(*
  A start position detection function block dummy.
  A dummy implementation to simulate start triggers at desired positions.
*)
FUNCTION_BLOCK FB_StartPositionDummy EXTENDS FB_BasePrint IMPLEMENTS I_StartPosDetect, I_PrintStatusClient, I_Simulation
VAR_INPUT
  bTrigger                    : BOOL;       // manual trigger
  lPosition                   : DINT;       // current position [SubPx]
  fSpeed                      : LREAL;      // current speed [m/s]
  fResolution                 : LREAL;      // current print resolution [dpi*SubPx]
END_VAR

VAR
  // properties
  _bSim               : BOOL;       // simulatio mode active (PROPERTY)
  _bCreateTrigger     : BOOL;       // create new CT trigger (PROPERTY)
  _nStartPosX0        : DINT;       // create position for CT (absolut) [SubPx] (PROPERTY)
  _bAutoTrigger       : BOOL;       // automatic sheet triggers
  
  // config
  iJobDefinition      : CalmarCompPrint.I_JobDefinition;
  
  // local helper
  rfNewCT             : RF_TRIG;    // trigger new ct
  nSheetLength        : DINT;       // sheet length in [SubPx]
  nSheetGap           : DINT;       // sheet gap in [SubPx]
  nSheetEndPosition   : DINT;       // sheet end position [SubPx]
  nNextSheetPosition  : DINT;       // next trigger location
  fSheetPerHour       : LREAL;      // sheets per hour
  fSheetSpeed         : LREAL;      // [m/min] speed meter per minute
  tCheckTrigger       : TON;
  
  tCurrentTimeStamp   : T_DCTIME64; // get current timestamp
  fCurrentTimeStamp   : LREAL;      // current timestamp
  fSensorTimeStamp    : LREAL;      // sensor timestamp
  fDeltaDistance      : LREAL;      // distance that the substrate moved between the detection and the treatment of the information [m]
END_VAR

VAR PERSISTENT
  // simulation configuration
  fSheetLength   : LREAL := 0.5;    // [m] sheet length (local or per job given)
  fSheetGap      : LREAL := 0.12;   // [m] gap between two sheets
END_VAR

// checks and fixes
IF iJobDefinition = 0 THEN RETURN; END_IF
IF NOT _bSim THEN RETURN; END_IF
IF fSpeed = 0 THEN RETURN; END_IF
IF fSheetLength = 0 THEN fSheetLength := 1; END_IF
IF fResolution = 0 THEN fResolution := 600*32; END_IF

// calculations
fSheetSpeed := fSpeed * 60;  // [m/s] -> [m/min]
nSheetGap := F_MeterToSubPixel(fPosMeter := fSheetGap, fResoSubPx := fResolution);  // [m] -> [SubPx]
fSheetPerHour := (60*60)/((fSheetLength+fSheetGap)/fSpeed);
nSheetLength := F_MeterToSubPixel(fPosMeter := fSheetLength, fResoSubPx := fResolution);  // [mm] -> [SubPx]
nNextSheetPosition := _nStartPosX0 + nSheetLength + nSheetGap; 
tCheckTrigger(PT:=TO_TIME(((fSheetLength+fSheetGap)/fSpeed)*1000));

// internal trigger creation
IF (lPosition - nNextSheetPosition) > 0 AND _bAutoTrigger THEN
  bTrigger := TRUE;
  tCheckTrigger(IN:=FALSE);
  tCheckTrigger(IN:=TRUE);
END_IF

// on trigger
rfNewCT(CLK := bTrigger, RT => _bCreateTrigger);
IF _bCreateTrigger THEN   // new ct created
  bTrigger := FALSE;  // reset trigger
  
  (* Calculate the current and sensor time stamp (keep old code not really necessary because we use current timestamp)*)
  tCurrentTimeStamp := F_GetCurDcTaskTime64();
  fCurrentTimeStamp := (ULINT_TO_LREAL(tCurrentTimeStamp )) / 1_000_000.0; (*in ms*)
  fSensorTimeStamp  := fCurrentTimeStamp;
  fDeltaDistance := (fCurrentTimeStamp - fSensorTimeStamp) * 0.001 * fSpeed;  (*Distance that the substrate moved between the detection and the treatment of the information [m]*)
  
  // sheet start and sheet end pos in [SubPx]
  _nStartPosX0     := lPosition - F_MeterToSubPixel(fPosMeter := fDeltaDistance, fResoSubPx := fResolution);
  nSheetEndPosition := _nStartPosX0 + nSheetLength;
END_IF

PROPERTY bSimEnable : BOOL
GET
bSimEnable := _bSim;
END_GET
SET
_bSim := bSimEnable;
END_SET
END_PROPERTY

(*
  A new container detected.
  NOTE: a pulse only
*)
PROPERTY bStartTrig : BOOL
GET
bStartTrig := _bCreateTrigger;
END_GET
END_PROPERTY

(*
  A valid container detected.
*)
PROPERTY bValid : BOOL
GET
bValid := TRUE;
END_GET
END_PROPERTY

METHOD mJobPause
END_METHOD

METHOD mJobStart
VAR_INPUT
	sJobDef	: CalmarCompPrint.I_JobDefinition;
END_VAR
IF sJobDef = 0 THEN LogError('JobStart: no sJobDef given'); RETURN; END_IF

iJobDefinition := sJobDef;    // current job definition
fSheetLength := iJobDefinition.fSubstrateDepth;
END_METHOD

METHOD mJobStop
VAR_INPUT
	sStatus	: CalmarCompPrint.I_JobStatus;
END_VAR
iJobDefinition := 0;    // delete job definition
END_METHOD

METHOD mProduced
VAR_INPUT
	(* current progress*)
	sProgress	: CalmarCompPrint.I_JobProgress;
END_VAR
; // nothing to do
END_METHOD

(*
  Detected start position X0 (absolute) in [SubPx].
*)
PROPERTY nStartPositionX0 : DINT
GET
nStartPositionX0 := _nStartPosX0;
END_GET
END_PROPERTY

METHOD SimEnter : BOOL
LogInfo('Enter start position creator simulation');
_bSim := TRUE;

_nStartPosX0 := lPosition;
nSheetEndPosition := lPosition;
nNextSheetPosition := lPosition;
END_METHOD

METHOD SimExit : BOOL
LogInfo('Exit start position creator simulation');
_bSim := FALSE;
END_METHOD

METHOD SimUpdate : BOOL
; // nothing to do
END_METHOD

END_FUNCTION_BLOCK

(* stored: Version 1.1.0.1, ProductVersion 3.1.4024.11
   POU FB_StartPositionDummy: Id {8c44436b-fdf6-4982-bb45-487571d5b646}, SpecialFunc None
   Folder I_PrintStatusClient: Id {0f059572-48fa-432b-b785-512422fd1dfe}
   Folder I_Simulation: Id {7d61ad54-78ed-4583-824e-3b28cb4bdfce}
   Folder I_StartPosDetect: Id {42dcb401-5898-4788-a131-7c35bf2d9f5b}
   Property bSimEnable: Id {9ad55ae0-9c7f-42e0-b227-356775d240a7}
   Get Get: Id {9bd88754-a865-4550-9123-bca0f19be00e}
   Set Set: Id {b66c4a74-41e4-4373-95c4-8e6dd06c2d09}
   Property bStartTrig: Id {3a919c9a-ce16-49c6-b57e-75dcd07db7d1}
   Get Get: Id {0a392f0b-d23a-4374-a637-12c72e002d9f}
   Property bValid: Id {dd397979-b437-4cd6-bdee-6dad5733a67f}
   Get Get: Id {7761d967-0a1f-4e88-ad34-4ad5ce416735}
   Method mJobPause: Id {7eb46286-2488-433d-8cdd-400aef51086a}
   Method mJobStart: Id {e393908f-23a1-4595-a465-2cf3c9f6001e}
   Method mJobStop: Id {d8356075-2335-4b08-acc5-155ab282c68f}
   Method mProduced: Id {fe7716e6-798e-41d7-838b-f7b407401b42}
   Property nStartPositionX0: Id {6b27a535-635b-4868-a381-d2f4a2a26ba0}
   Get Get: Id {1b86c0b7-703e-4025-917d-2f98f1c0050d}
   Method SimEnter: Id {5f3afcf0-45e7-43f3-b7fa-173569233158}
   Method SimExit: Id {48b25644-8173-4c12-af95-8aee36151a4f}
   Method SimUpdate: Id {8e513948-d863-4b3f-8f45-576ad340d53b} *)
